// TIA Portal V15.1 export
// export: Created 2026-01-15T16:29:48.7488975Z, ExportSetting WithDefaults, WithReadOnly, DisplayName Totally Integrated Automation Portal, DisplayVersion V15.1 Update 8, DisplayName TIA Portal Openness, DisplayVersion V15.1 Update 8, DisplayName STEP 7 Professional, DisplayVersion V15.1 Update 8, DisplayName WinCC Advanced, DisplayVersion V15.1 Update 8
DATA_BLOCK "PLC_BIT"   // DB9
{ S7_Optimized_Access := 'FALSE' }
VERSION : 0.1
// stored: AutoNumber true, CodeModifiedDate 2026-01-01T12:46:58.5268647Z, CompileDate 2026-01-15T16:25:48.0586708Z, CreationDate 2026-01-15T16:24:02.4619467Z, DBAccessibleFromOPCUA true, InterfaceModifiedDate 2026-01-01T12:46:58.5268647Z, IsConsistent true, IsKnowHowProtected false, IsOnlyStoredInLoadMemory false, IsPLCDB false, IsWriteProtectedInAS false, ModifiedDate 2026-01-12T10:28:53.5688727Z, ParameterModified 2026-01-01T12:46:58.5268647Z, StructureModified 2026-01-01T12:46:58.5268647Z
   VAR
      RUN : Bool;
      MAN : Bool;
      AUT : Bool;
      SIM : Bool;
      PAU : Bool;
      NTR_FU : Bool;   // Nồi trộn đã đượcnạp đầy
      PCH_FU : Bool;
      SKIP_FU : Bool;
      AGG1_FU : Bool;   // Silo AGG1 Full
      WAG1_FU : Bool;   // Cân AG1 Full
      WAG1_EM : Bool;   // Cân AG1 Empty
      AGG2_FU : Bool;   // Silo AGG2 Full
      WAG2_FU : Bool;   // Cân AG2 Full
      WAG2_EM : Bool;   // Cân AG2 Empty
      AGG3_FU : Bool;   // Silo AGG3 Full
      WAG3_FU : Bool;   // Cân AG3 Full
      WAG3_EM : Bool;   // Cân AG3 Empty
      AGG4_FU : Bool;   // Silo AGG4 Full
      WAG4_FU : Bool;   // Cân AG4 Full
      WAG4_EM : Bool;   // Cân AG4 Empty
      AGG5_FU : Bool;   // Silo AGG5 Full
      WAG5_FU : Bool;   // Cân AG5 Full
      WAG5_EM : Bool;   // Cân AG5 Empty
      AGG6_FU : Bool;   // Silo AGG6 Full
      WAG6_FU : Bool;   // Cân AG6 Full
      WAG6_EM : Bool;   // Cân AG6 Empty
      CEM1_FU : Bool;   // Silo CEM/FD1 Full
      CEM2_FU : Bool;   // Silo CEM/FD2 Full
      CEM3_FU : Bool;   // Silo CEM/FD3 Full
      WCE1_FU : Bool;   // Cân CE/FD1 Full
      WCE1_EM : Bool;   // Cân CE/FD1 Empty
      CEM4_FU : Bool;   // Silo CEM/FD4 Full
      CEM5_FU : Bool;   // Silo CEM/FD5 Full
      WCE2_FU : Bool;   // Cân CE/FD2 Full
      WCE2_EM : Bool;   // Cân CE/FD2 Empty
      WAT1_FU : Bool;   // Weigh Asphalt Tank 1 Full - Cảm biến báo bể nhựa 1 đầy
      WWA1_FU : Bool;   // Weigh Water Asphalt 1 Full - Cảm biến báo phễu cân nhựa 1 đầy
      WWA1_EM : Bool;   // Weigh Water Asphalt 1 Empty - Cảm biến báo phễu cân nhựa 1 rỗng
      WAT2_FU : Bool;   // Weigh Asphalt Tank 2 Full - Cảm biến báo bể nhựa 2 đầy
      WWA2_FU : Bool;   // Weigh Water Asphalt 2 Full - Cảm biến báo phễu cân nhựa 2 đầy
      WWA2_EM : Bool;   // Weigh Water Asphalt 2 Empty - Cảm biến báo phễu cân nhựa 2 rỗng
      ADD1_FU : Bool;   // Silo phụ gia 1 Full
      ADD2_FU : Bool;   // Silo phụ gia 2 Full
      ADD3_FU : Bool;   // Silo phụ gia 3 Full
      WAD1_FU : Bool;   // Cân phụ gia 1 Full
      WAD1_EM : Bool;   // Cân phụ gia 1 Empty
      ADD4_FU : Bool;   // Silo phụ gia 4 Full
      ADD5_FU : Bool;   // Silo phụ gia 5 Full
      ADD6_FU : Bool;   // Silo phụ gia 6 Full
      WAD2_FU : Bool;   // Cân phụ gia 2 Full
      WAD2_EM : Bool;   // Cân phụ gia 2 Empty
      "BAT/TAT NT" : Bool;   // Bật tắt băng tải ngang
      "BAT/TAT BTX" : Bool;   // Bật tắt băng tải xiên
      "NN_CAN NUOC" : Bool;
      "NN_XA NUOC" : Bool;
      NN_MCN : Bool;
      NN_DCN : Bool;
      "NN_DONG KEP" : Bool;
      "NN_MO KEP" : Bool;
      "NN_GAU LEN" : Bool;
      "NN_DUNG GAU" : Bool;
      "NN_GAU XUONG" : Bool;
      TOP_BTC : Bool;
      "TOP. GAU LEN" : Bool;
      "TOP. GAU XUONG" : Bool;
      "COT LIEU_FU" : Bool;
      PCĐ_SIM : Bool;
      PCM_SIM : Bool;
      CNĐ_SIM : Bool;
      CNM_SIM : Bool;
      "CN1/2_SIM" : Bool;
      COT_LIEU_FU : Bool;
      KT_XA_AGG : Bool;
      NEXT_WAGG1 : Bool;
      NEXT_WAGG2 : Bool;
      NEXT_WAGG3 : Bool;
      NEXT_WAGG4 : Bool;
      NEXT_WAGG5 : Bool;
      NEXT_WAGG6 : Bool;
      NEXT_WCEM1 : Bool;   // Nếu SV_FD1=0 thì bỏ qua Cân FD1
      NEXT_WCEM2 : Bool;
      NEXT_WWAT1 : Bool;
      NEXT_WWAT2 : Bool;
      NEXT_WADD1 : Bool;
      NEXT_WADD2 : Bool;
      End_Agg1 : Bool;
      End_Agg2 : Bool;
      End_Agg3 : Bool;
      End_Agg4 : Bool;
      End_Agg5 : Bool;
      End_Agg6 : Bool;
      SW_MODE : Bool;
   END_VAR
BEGIN
END_DATA_BLOCK
